(* PLC project static_torsion.project, CODESYS CODESYS V3.5 SP17 Patch 3 *)
(* stored: creationDateTime 1970-01-01T00:00:00, modificationDateTime 2026-06-22T15:12:39.4699931 *)

FUNCTION_BLOCK SERVO
  VAR
    xPowerStatus : BOOL;
    fbPower : MC_Power;
    fbStop : MC_Stop;
    fbHalt : MC_Halt;
    fbFollow : SMC_FollowVelocity;
    fbMoveRel : MC_MoveRelative;
    fbJog : MC_Jog;
    fbReset : MC_Reset;
    fbActualVelocity : MC_ReadActualVelocity;
    fbStatus : MC_ReadStatus;
    iDriveStatus : INT;
    xPowerEnable : BOOL := TRUE;
    prevCommand_ID : CTRL_ID;
    xReset : BOOL;
    xPIDStart : BOOL;
    lrSpeed : LREAL := 0;
    xHalt : RS;
    xStop : BOOL;
    xJogForward : BOOL;
    xJogBackward : BOOL;
    lrJogVelocity : LREAL;
  END_VAR

            //
fbPower(Axis:= MainDrive, Enable:= TRUE);
fbStop(Axis:= MainDrive);
fbHalt(Axis:= MainDrive, Deceleration := 1000, Jerk:= 10000);
fbFollow(Axis:= MainDrive);
fbMoveRel(Axis := MainDrive);
fbJog(Axis := MainDrive, Acceleration:= 1000, Deceleration:= 1000, Jerk:= 10000);
fbReset(Axis := MainDrive);

iDriveStatus := MainDrive.nAxisState;
fbActualVelocity(Axis:= MainDrive, Enable:= TRUE);
fbStatus(Axis:= MainDrive, Enable:= TRUE);

lrJogVelocity := TO_LREAL(GVL.iJogVelocity)/10.0;
          

ACTION POWER_OFF:
                fbPower.bRegulatorOn	:= FALSE;
fbPower.bDriveStart		:= FALSE;

fbJog.JogForward 		:= FALSE;
fbJog.JogBackward		:= FALSE;
fbJog.Velocity			:= 0.0;

              
END_ACTION

ACTION POWER_ON:
                fbPower.bRegulatorOn:= TRUE;
fbPower.bDriveStart:= TRUE;
              
END_ACTION

ACTION HALT:
                fbJog.JogForward		:= FALSE;
fbJog.JogBackward		:= FALSE;
fbJog.Velocity			:= 0.0;

fbFollow.bExecute		:= FALSE;
fbFollow.fSetVelocity	:= 0.0;

fbHalt.Execute			:= TRUE;

xReset := FALSE;
xPIDStart := FALSE;
xJogForward := xJogBackward := FALSE;
xHalt.RESET1 := FALSE;
xHalt.SET := TRUE;
lrSpeed := 0.0;
              
END_ACTION

ACTION JOG_CW:
                fbHalt.Execute		:= FALSE;
fbJog.JogForward	:= TRUE;
fbJog.JogBackward	:= FALSE;
fbJog.Velocity		:= lrJogVelocity;

              
END_ACTION

ACTION JOG_CCW:
                fbHalt.Execute		:= FALSE;
fbJog.JogForward	:= FALSE;
fbJog.JogBackward	:= TRUE;
fbJog.Velocity		:= lrJogVelocity;
              
END_ACTION

ACTION TORQUE_HOLD:
                fbHalt.Execute			:= FALSE;
fbJog.JogForward		:= FALSE;
fbJog.JogBackward		:= FALSE;
fbJog.Velocity			:= 0.0;

fbFollow.bExecute		:= TRUE;
fbFollow.fSetVelocity	:= GVL.lrFollowVelocity;


              
END_ACTION

ACTION MOVE_TO_ANGLE:
                
              
END_ACTION

METHOD RESET_ERROR : SMC_ERROR
  VAR_INPUT
    Execute : BOOL;
  END_VAR
                  fbReset.Execute := Execute;
RESET_ERROR := fbReset.ErrorID;
                
END_METHOD
END_FUNCTION_BLOCK
